# EPICS substitutions: doc/EXAMPLE_bsread.subs
# Macros:
# P  -  Record prefix, e.g. MTEST-HW3-R

file bsread.template {
	{
		P = "MTEST-HW3-R"
	}
}
